TYPE E_InstrumentEnergyType :
(
	InstruType_isNull := 0,
	InstruType_isMonopole := 1,
	InstruType_isBipolar := 2,
	InstruType_isUltraKnife := 3,
	InstruType_isForceBipolar := 5
);
END_TYPE

(* stored: Version 1.1.0.1, ProductVersion 3.1.4024.11
   DUT E_InstrumentEnergyType: Id {fa30c82e-55d5-44ce-9ee5-7c02a2e0549f} *)
